// TwinCAT 3 PLC project Untitled1
// ProgramVersion: 3.1.4024.0
// libraries:
//   CmpBitmapPool, * (System)
//   Tc2_Standard, * (Beckhoff Automation GmbH)
//   Tc2_System, * (Beckhoff Automation GmbH)
//   Tc3_Module, * (Beckhoff Automation GmbH)
//   VisuDialogs, * (System)
// project tree:
//   / GlobalTextList.TcGTLO, PlcTask.TcTTO, Visualization Manager.TcVMO (not stored)
//   GVLs/ GVL_hesapSayfa.TcGVL, GVL_Mesai_Ucret.TcGVL, GVL_uye_panel.TcGVL, GVL_mesai_gun.TcGVL, GVL_mesai_saat.TcGVL, GVL_personel_kayit.TcGVL
//   POUs/ ImagePool.TcIPO (not stored), MAIN.TcPOU, POU_2.TcPOU
//   VISUs/ Hesap_Sayfa.TcVIS, Kayit_Sayfa.TcVIS, mesaigunleri_sayfa.TcVIS, MesaiSaat_sayfa.TcVIS, uyelik_sayfa.TcVIS, Ana_Sayfa.TcVIS
// real-time tasks:
//   TASK PlcTask: cycle T#10ms, priority 20, ADS port 350

CONFIGURATION Untitled1
    RESOURCE PLC ON TwinCAT3
        TASK PlcTask(INTERVAL := T#10ms, PRIORITY := 20);
        PROGRAM MAIN WITH PlcTask : MAIN;
    END_RESOURCE
END_CONFIGURATION

// ---- GVLs/GVL_hesapSayfa.TcGVL
{attribute 'qualified_only'}
VAR_GLOBAL
	

saydir1: TON;
start:BOOL;
cikis:BOOL;
gecensure:TIME;
gecenzaman:INT;
hesaplama:INT;






END_VAR

// ---- GVLs/GVL_Mesai_Ucret.TcGVL
{attribute 'qualified_only'}
VAR_GLOBAL
	

hesapla:INT;
mesaiUcret:INT;
online:BOOL;
kaydet:BOOL;






END_VAR

// ---- GVLs/GVL_uye_panel.TcGVL
{attribute 'qualified_only'}
VAR_GLOBAL
	








END_VAR

// ---- GVLs/GVL_mesai_gun.TcGVL
{attribute 'qualified_only'}
VAR_GLOBAL
	
pazartesi:BOOL;
sali:BOOL;
carsamba:BOOL;
persembe:BOOL;
cuma:BOOL;
cumartesi:BOOL;
pazar:BOOL;
kaydet:BOOL;


END_VAR

// ---- GVLs/GVL_mesai_saat.TcGVL
{attribute 'qualified_only'}
VAR_GLOBAL
	

kaydet:BOOL;
i:INT;
baslangicDk:INT;
bitisDk:INT;
baslangicSn:INT;
bitisSn:INT;
cikis:BOOL;
sayac:INT;
sayac1:INT;
j:INT;
sayac2:INT;
n:INT;
sayac3:INT;
h:INT;
mesaiucret:INT;
saat:INT;
mesaiSaaat:INT;



x1_mesaiSaat:INT;
x1_5mesaiSaat:REAL;
x_3mesaiSaat:REAL;
tum_mesai:REAL;




x1_5baslangicSaat : INT;
x_3baslangicSaat:INT;




x1bslangicSaat:INT;
x1bslangicdakika:INT;
x1bitisSaat:INT;
x1bitisdakika:INT;



x1_5bslangicSaat:INT;
x1_5bslangicdakika:INT;
x1_5bitisSaat:INT;
x1_5bitisdakika:INT;




x3bslangicSaat:INT;
x3bslangicdakika:INT;
x3bitisSaat:INT;
x3bitisdakika:INT;










baslangicdakika: STRING;
baslangicsaat: STRING;
bitisdakika: STRING;
bitissaat: STRING;




a:BOOL;
b:BOOL;
c:BOOL;
d:BOOL;
e:BOOL;
f:BOOL;






































END_VAR

// ---- GVLs/GVL_personel_kayit.TcGVL
{attribute 'qualified_only'}
VAR_GLOBAL
	

perid:STRING;
perisim:STRING;
perSoyisim:STRING;

perMesaiGun:BOOL;
perMesaiSaat:BOOL;

kaydet:BOOL;
msgtype:MESSAGEBOXDIALOG_TYPES;
messagetitle:STRING;
messagetext:STRING;
cikis3:BOOL;
sayac:INT;
i:INT := 1;
sayac1:INT;
j:INT;
sayac2:INT;
g:INT;



dogru : BOOL;
invisibleKayit : BOOL;





personelisim:ARRAY[1..70] OF STRING;
personelsoyisim:ARRAY[1..70] OF STRING;
personelid:ARRAY[1..70] OF STRING;






saydirici:R_TRIG ;



temizle:BOOL;
















END_VAR

// ---- POUs/MAIN.TcPOU
PROGRAM MAIN
VAR
	



isim:ARRAY[0..70] OF STRING;
kullanici: ARRAY[0..70] OF STRING;
sifreler: ARRAY[0..70] OF STRING;
soyisim:ARRAY[0..70] OF STRING;
gunler:ARRAY[1..7] OF BOOL;

ad:STRING;
soyad:STRING;
kuladi:STRING;
sifre:STRING;

kaydet:BOOL;







uyelik:BOOL;
uyelik1:BOOL;
sayici:INT;



giris:BOOL;




yenikul:STRING;
yenisifre:STRING;





msgtype:MESSAGEBOXDIALOG_TYPES;
msgtitle:STRING;
msgtxt:STRING;



i: INT;
j:INT;
	
	cikis: BOOL;
	

	

	saydir: R_TRIG;
	cikis2: BOOL;
	sayici1: INT;
	kaydet2: BOOL;
	sayici2: INT;
	g: INT;
	sayici3: INT;
	h: INT;
	n: INT;
	giris1: BOOL;
	
	mesai_saat_saydirici: R_TRIG;
	
END_VAR



msgtitle:='İşlem Durumu ';
msgtxt:='Kayıt İşlemi Başarılı..';


GVL_personel_kayit.messagetext:='Kayıt İşlemi Başarılı.. Mesai Ücreti Hesaplamak Mesai Günü Seç  Butonuna Basınız.';
GVL_personel_kayit.messagetitle:='Kayıt İşlemi Durumu';






Giris_Panel();
uyelik_panel();
Kayit_Sayfa();
mesai_gun();
mesai_saat();
Hesap_Panel();

ACTION Giris_Panel:

giris1:=FALSE;

IF GVL_personel_kayit.perMesaiGun THEN
	GVL_personel_kayit.dogru:=TRUE;
	
END_IF


IF giris=TRUE THEN
	
FOR n:=1 TO 70 BY 1 DO
	
  IF kullanici[n]=kuladi AND sifreler[n]=sifre AND NOT GVL_personel_kayit.dogru THEN
	  
 
	  VisuElems.CurrentVisu := 'Kayit_Sayfa';
	  
	  
	  
	 
  END_IF

  	
END_FOR

	
END_IF
END_ACTION

ACTION Hesap_Panel:

GVL_mesai_saat.mesaiucret:=50;
GVL_hesapSayfa.saydir1(IN:=GVL_hesapSayfa.start , PT:=T#10S , Q=>GVL_hesapSayfa.cikis , ET=>GVL_hesapSayfa.gecensure );

GVL_hesapSayfa.start:=TRUE;



IF GVL_hesapSayfa.cikis=TRUE THEN
	
 IF 
	 GVL_mesai_gun.pazartesi=TRUE  OR  GVL_mesai_gun.sali=TRUE OR  GVL_mesai_gun.carsamba=TRUE OR  GVL_mesai_gun.persembe=TRUE OR  GVL_mesai_gun.cuma=TRUE THEN
	
	
(*   IF GVL_mesai_saat.baslangicsaat < GVL_mesai_saat.bitissaat  THEN
    	GVL_hesapSayfa.hesaplama:= GVL_mesai_saat.bitissaat-GVL_mesai_saat.baslangicsaat;
		ELSE			
		GVL_hesapSayfa.hesaplama:=GVL_mesai_saat.baslangicsaat-GVL_mesai_saat.bitisdakika;
		
 
 
END_IF
 *)
	
	
	
 
 END_IF
 
 
 
 

 
(*  IF GVL_mesai_gun.cumartesi OR GVL_mesai_gun.pazar THEN
	 	
   	 
 GVL_hesapSayfa.hesaplama:= GVL_mesai_saat.bitisdakika-GVL_mesai_saat.baslangicdakika;
 
 
 END_IF
 *)
 
 
 



	
END_IF
END_ACTION

ACTION Kayit_sayfa:


GVL_personel_kayit.saydirici(CLK:=GVL_personel_kayit.kaydet , Q=>GVL_personel_kayit.cikis3 );

IF GVL_personel_kayit.kaydet THEN
	GVL_personel_kayit.invisibleKayit:=TRUE;
END_IF

IF VisuElems.CurrentVisu='mesaigunleri_sayfa'THEN
	GVL_personel_kayit.invisibleKayit:=FALSE;
END_IF


IF GVL_personel_kayit.kaydet=TRUE THEN
	
IF GVL_personel_kayit.cikis3=TRUE THEN
 
GVL_personel_kayit.sayac:=GVL_personel_kayit.sayac +1;

END_IF



FOR GVL_personel_kayit.i:=1 TO 70 BY 1 DO
	
IF GVL_personel_kayit.personelisim[GVL_personel_kayit.i] ='' THEN
	GVL_personel_kayit.personelisim[GVL_personel_kayit.i]:=GVL_personel_kayit.perisim;
		
ELSE
	GVL_personel_kayit.personelisim[GVL_personel_kayit.sayac]:=GVL_personel_kayit.perisim;
	
END_IF

EXIT;
END_FOR






IF GVL_personel_kayit.cikis3=TRUE THEN
	
	GVL_personel_kayit.sayac1:=GVL_personel_kayit.sayac1+1;		
END_IF

FOR GVL_personel_kayit.j:=1 TO 70 BY  1 DO
	
IF GVL_personel_kayit.personelsoyisim[GVL_personel_kayit.j]='' THEN
	GVL_personel_kayit.personelsoyisim[GVL_personel_kayit.j]:=GVL_personel_kayit.perSoyisim;
	ELSE
		GVL_personel_kayit.personelsoyisim[GVL_personel_kayit.sayac]:=GVL_personel_kayit.perSoyisim;
	
END_IF

EXIT;

END_FOR



IF GVL_personel_kayit.cikis3=TRUE THEN
	GVL_personel_kayit.sayac2:=GVL_personel_kayit.sayac2 +1;
	
END_IF

FOR GVL_personel_kayit.g:=1 TO 70 BY 1 DO
	
	IF GVL_personel_kayit.personelid[GVL_personel_kayit.g]='' THEN
		GVL_personel_kayit.personelid[GVL_personel_kayit.g]:=GVL_personel_kayit.perid;
		ELSE
		GVL_personel_kayit.personelid[GVL_personel_kayit.sayac2]:=GVL_personel_kayit.perid;	
		
	END_IF
	EXIT;
	
END_FOR



















END_IF




IF GVL_personel_kayit.temizle=TRUE THEN
	GVL_personel_kayit.perisim:='';
	GVL_personel_kayit.perSoyisim:='';
	GVL_personel_kayit.perid:='';
	
	
	
	


END_IF
END_ACTION

ACTION mesai_gun:





IF GVL_mesai_gun.pazartesi=TRUE THEN
	
	
GVL_mesai_gun.sali:=FALSE;
GVL_mesai_gun.carsamba:=FALSE;
GVL_mesai_gun.persembe:=FALSE;
GVL_mesai_gun.cuma:=FALSE;
GVL_mesai_gun.cumartesi:=FALSE;
GVL_mesai_gun.pazar:=FALSE;


END_IF






IF GVL_mesai_gun.sali=TRUE THEN
	
	
GVL_mesai_gun.pazartesi:=FALSE;
GVL_mesai_gun.carsamba:=FALSE;
GVL_mesai_gun.persembe:=FALSE;
GVL_mesai_gun.cuma:=FALSE;
GVL_mesai_gun.cumartesi:=FALSE;
GVL_mesai_gun.pazar:=FALSE;


END_IF





IF GVL_mesai_gun.carsamba=TRUE THEN
	
	
GVL_mesai_gun.pazartesi:=FALSE;
GVL_mesai_gun.sali:=FALSE;
GVL_mesai_gun.persembe:=FALSE;
GVL_mesai_gun.cuma:=FALSE;
GVL_mesai_gun.cumartesi:=FALSE;
GVL_mesai_gun.pazar:=FALSE;


END_IF




IF GVL_mesai_gun.persembe=TRUE THEN
	
	
GVL_mesai_gun.pazartesi:=FALSE;
GVL_mesai_gun.sali:=FALSE;
GVL_mesai_gun.carsamba:=FALSE;
GVL_mesai_gun.cuma:=FALSE;
GVL_mesai_gun.cumartesi:=FALSE;
GVL_mesai_gun.pazar:=FALSE;


END_IF





IF GVL_mesai_gun.cuma=TRUE THEN
	
	
GVL_mesai_gun.pazartesi:=FALSE;
GVL_mesai_gun.sali:=FALSE;
GVL_mesai_gun.carsamba:=FALSE;
GVL_mesai_gun.persembe:=FALSE;
GVL_mesai_gun.cumartesi:=FALSE;
GVL_mesai_gun.pazar:=FALSE;


END_IF






IF GVL_mesai_gun.cumartesi=TRUE THEN
	
	
GVL_mesai_gun.pazartesi:=FALSE;
GVL_mesai_gun.sali:=FALSE;
GVL_mesai_gun.carsamba:=FALSE;
GVL_mesai_gun.persembe:=FALSE;
GVL_mesai_gun.cuma:=FALSE;
GVL_mesai_gun.pazar:=FALSE;


END_IF
IF GVL_mesai_gun.pazar=TRUE THEN
	
	
GVL_mesai_gun.pazartesi:=FALSE;
GVL_mesai_gun.sali:=FALSE;
GVL_mesai_gun.carsamba:=FALSE;
GVL_mesai_gun.persembe:=FALSE;
GVL_mesai_gun.cumartesi:=FALSE;
GVL_mesai_gun.cuma:=FALSE;


END_IF
END_ACTION

ACTION mesai_saat:



GVL_mesai_saat.a:=FALSE;
GVL_mesai_saat.b:=FALSE;
GVL_mesai_saat.c:=FALSE;




 // Başlangıç Dakikası
IF GVL_mesai_saat.kaydet=TRUE THEN
	

	 
  
	IF GVL_mesai_saat.x1bslangicSaat>GVL_mesai_saat.x1bitisSaat THEN
	
	GVL_mesai_saat.x1_mesaiSaat:=GVL_mesai_saat.x1bslangicSaat-GVL_mesai_saat.x1bitisSaat;
	GVL_mesai_saat.a:=TRUE;
	ELSE
		
	GVL_mesai_saat.x1_mesaiSaat:=GVL_mesai_saat.x1bitisSaat-GVL_mesai_saat.x1bslangicSaat;
	GVL_mesai_saat.b:=TRUE;
	
	END_IF
 



	IF GVL_mesai_saat.x1_5bslangicSaat>GVL_mesai_saat.x1_5bitisSaat THEN
	
	GVL_mesai_saat.x1_5mesaiSaat:=(GVL_mesai_saat.x1_5bslangicSaat-GVL_mesai_saat.x1_5bitisSaat)*1.5;
	GVL_mesai_saat.c:=TRUE;
	
	ELSE
		
	
	GVL_mesai_saat.x1_5mesaiSaat := (GVL_mesai_saat.x1_5bitisSaat-GVL_mesai_saat.x1_5bslangicSaat)*1.5;
	GVL_mesai_saat.d:=TRUE;
	
	END_IF


	
     
	 




	IF GVL_mesai_saat.x3bslangicSaat>GVL_mesai_saat.x3bitisSaat THEN
	
	GVL_mesai_saat.x_3mesaiSaat:=(GVL_mesai_saat.x3bslangicSaat-GVL_mesai_saat.x3bitisSaat)*3;
	GVL_mesai_saat.e:=TRUE;
	ELSE
		
	GVL_mesai_saat.x_3mesaiSaat:=(GVL_mesai_saat.x3bitisSaat-GVL_mesai_saat.x3bslangicSaat)*3;
	GVL_mesai_saat.f:=TRUE;
	
	END_IF
	
	
	
	
	
	IF GVL_mesai_saat.a=TRUE  OR GVL_mesai_saat.b=TRUE  THEN
		GVL_mesai_saat.mesaiSaaat:=GVL_mesai_saat.x1_mesaiSaat;
		
	END_IF
	
	
	
	(* IF GVL_mesai_saat.c=TRUE  OR GVL_mesai_saat.d=TRUE  THEN
		
		GVL_mesai_saat.mesaiSaaat:=GVL_mesai_saat.x1_5mesaiSaat;
	END_IF
	
	IF GVL_mesai_saat.e=TRUE OR GVL_mesai_saat.f=TRUE THEN
		
		GVL_mesai_saat.mesaiSaaat:=GVL_mesai_saat.x_3mesaiSaat;
	END_IF *)
	
	GVL_mesai_saat.tum_mesai:=(GVL_mesai_saat.x1_mesaiSaat+GVL_mesai_saat.x1_5mesaiSaat+GVL_mesai_saat.x_3mesaiSaat);
 
	
	
	


END_IF
END_ACTION

ACTION Mesai_Ucret_Panel:



GVL_Mesai_Ucret.online:=TRUE;
END_ACTION

ACTION uyelik_panel:


saydir(CLK:=kaydet , Q=>cikis );
		
		

IF kaydet=TRUE THEN




IF cikis=TRUE THEN
	sayici:=sayici+1;
END_IF

	FOR i:=1 TO 70 BY 1 DO
	
		IF isim[i]='' THEN			
			isim[i]:=ad;
		ELSE
			isim[sayici]:=ad;
		END_IF
		
		EXIT;
		
	END_FOR



IF cikis=TRUE THEN
	sayici1:=sayici1+1;
END_IF



FOR j:=1 TO 70 BY 1 DO
	
  IF soyisim[j]='' THEN
	  soyisim[j]:=soyad;
   ELSE
	soyisim[sayici1]:=soyad;
  END_IF


EXIT;
END_FOR










IF cikis=TRUE THEN
	sayici2:=sayici2+1;
	END_IF



FOR g:=1 TO 70 BY 1 DO
	
  IF kullanici[g]='' THEN
	  kullanici[g]:=yenikul;
	  ELSE
		  kullanici[sayici2]:=yenikul;
  END_IF


EXIT;
END_FOR







IF cikis=TRUE THEN
	sayici3:=sayici3+1;
	END_IF



FOR h:=1 TO 70 BY 1 DO
	
  IF sifreler[h]='' THEN
	  sifreler[h]:=yenisifre;
	  ELSE
		  sifreler[sayici3]:=yenisifre;
  END_IF


EXIT;
END_FOR


























	

END_IF
END_ACTION

END_PROGRAM

// ---- POUs/POU_2.TcPOU
PROGRAM POU_2
VAR
END_VAR

END_PROGRAM

// ---- GlobalTextList.TcGTLO
TEXTLIST GlobalTextList
  899 = '  '
  16 = '                          İsim:'
  1263 = '                   İsim:'
  435 = '                  İsim:'
  382 = '                İsim:'
  1202 = '             Soyisim:'
  479 = '            Soyisim:'
  1142 = '           Soyisim:'
  551 = '          Soyisim:'
  85 = '        Personel ID:'
  1102 = '       Personel ID:'
  510 = '      Personel ID:'
  1073 = '      Soyisim:'
  905 = '   Soyisim:'
  742 = '  Mesai Saati :'
  778 = '  Mesai Saati Seç'
  682 = ' Yeni Kullanıcı Adı :'
  954 = '%d'
  897 = '%d Saat Mesai Yapılmıştır'
  1058 = '%d Saat Mesai Yapılmıştır.'
  772 = '%d:%d'
  997 = '%ds'
  74 = '%s'
  388 = '%s:%s'
  62 = "%t[Son Güncelleme :'ddd MMM dd.MM.yy'at' HH:mm:ss]"
  507 = '-----------'
  528 = '------------------------'
  966 = '---------------------------'
  628 = '----------------------------'
  333 = '------------------------------'
  654 = '-----------------------------------'
  850 = '07:45'
  549 = '07:45/ 18:45'
  996 = '07:45/ 18:45 (X1)'
  963 = '07:45/ 18:45 (X1,5)'
  709 = '07:45/ 18:45 (X2)'
  404 = '07:45/ 18:45 (X2,5)'
  422 = '07:45/ 18:45 (X3)'
  728 = '0:%s'
  1004 = '1,5/X Mesai'
  1156 = '1/X Mesai'
  990 = '18:45/ 18:45 (X1)'
  1298 = '18:45/ 18:45 (X1,5)'
  471 = '18:45/ 23:45 (X1,5)'
  794 = '18:45/ 23:45 (X2)'
  1060 = '18:45/ 23:45 (X2,5)'
  900 = '23:45/ 07:45 (X2)'
  744 = '23:45/ 07:45 (X2,5)'
  436 = '23:45/ 07:45 (X3)'
  666 = '23:45/ 18:45 (X3)'
  885 = '23:45/07:45 (X3)'
  271 = '23:45/8:45 (X3)'
  892 = '3/X Mesai'
  919 = ':'
  653 = '@afşa'
  410 = 'Adı :'
  425 = 'Adınız           :'
  953 = 'Adınız       :'
  790 = 'Adınız   :'
  977 = 'Adınız  :'
  942 = 'Adınız :'
  176 = 'Afşa Robotik'
  1317 = 'Alacağı Ücret :'
  34 = 'Ana Sayfaya Dön'
  580 = 'ascascas'
  827 = 'asfqwfsvsdv'
  509 = 'Başlangıç :'
  773 = 'Başlangıç Saati :'
  1122 = 'Bilgilendirme'
  220 = 'Bitiş  Saati :'
  1442 = 'Bitiş :'
  817 = 'Bugünün Tarihni Giriniz :'
  252 = 'Bugünün Tariini Giriniz :'
  270 = 'Buugünün Tariini Giriniz :'
  683 = 'CUMA'
  325 = 'CUMARTESİ'
  241 = 'd'
  793 = 'G,n Sayfası'
  627 = 'Geriye Dön'
  1107 = 'Geriye Dön '
  318 = 'GERİYE DÖN'
  558 = 'Giriş'
  83 = 'Giriş Yap'
  994 = 'GroupBox'
  1049 = 'Gün Sayfası'
  301 = 'Gün Seç'
  1115 = 'Gün Çizelgesi'
  970 = 'GÜN ÇİZELGESİ'
  881 = 'GÜN/SAAT ÇİZELGESİ'
  984 = 'HAFTA SONU'
  965 = 'Hafta Sonu'
  323 = 'Hafta İçi'
  822 = 'HAFTA İÇİ'
  950 = 'Hesapla'
  472 = 'HESAPLANAN ÜCRET'
  860 = 'Isim :'
  546 = 'Kaydet'
  504 = 'KAYDET'
  501 = 'Kayıt Bilgisi'
  582 = 'Kullanıcı Adı'
  334 = 'Kullanıcı Adı :'
  995 = 'Label'
  188 = 'Mesai Gün Çizelgesi'
  39 = 'Mesai Günü'
  374 = 'Mesai Günü :'
  681 = 'Mesai Günü Seç'
  868 = 'Mesai Saati'
  298 = 'Mesai Saati :'
  918 = 'Mesai Saati : '
  281 = 'Mesai Saati Seç'
  788 = 'Mesai Saatini Giriniz :'
  256 = 'Mesai Ücreti'
  962 = 'Mesai Ücreti Hesapla'
  322 = 'MESAİ SAATİ UYGULAMASI'
  257 = 'OLUŞTUR'
  5 = 'PAZAR'
  819 = 'PAZARTESİ'
  293 = 'Personel Bilgileri'
  521 = 'Personel Bilgisi'
  799 = 'PERSONEL BİLGİSİ'
  514 = 'Personel ID:'
  752 = 'PERSONEL MESAİ TAKİP UYGULAMASI'
  129 = 'PERSONEL MESAİ-TAKİP'
  545 = 'Personel Soyisim :'
  512 = 'Personel İd'
  93 = 'Personel İd :'
  219 = 'Personel İsim :'
  731 = 'PERŞEMBE'
  140 = 'S'
  311 = 'saassacaxzc'
  506 = 'SALI'
  59 = 'sdasqwfqwf'
  508 = 'Soyadı :'
  810 = 'Soyadınız :'
  66 = 'Soyisim'
  847 = 'Soyisim :'
  910 = 'Soyisim:'
  581 = 'sOYİSİM:'
  336 = 'Temizle'
  20 = 'ullanıcı Adı :'
  1206 = 'x(1,5)'
  1002 = 'x(3)'
  655 = 'x1'
  1441 = 'x3'
  833 = 'YENİ KAYIT OLUŞTURMA'
  118 = 'YENİ ÜYE OLUŞTURMA'
  239 = 'Zamanı Giriniz :'
  476 = 'zxcZxc'
  299 = 'ÇARŞAMBA'
  452 = 'ÇIKIŞ'
  969 = 'Ücret :'
  602 = 'Üyelik Oluştur'
  937 = 'İsim      :'
  569 = 'İsim    :'
  614 = 'İsim  :'
  393 = 'İsim :'
  242 = 'İsim:'
  431 = 'Şifre'
  908 = 'Şifre :'
END_TEXTLIST

// ---- VISUs/Hesap_Sayfa.TcVIS
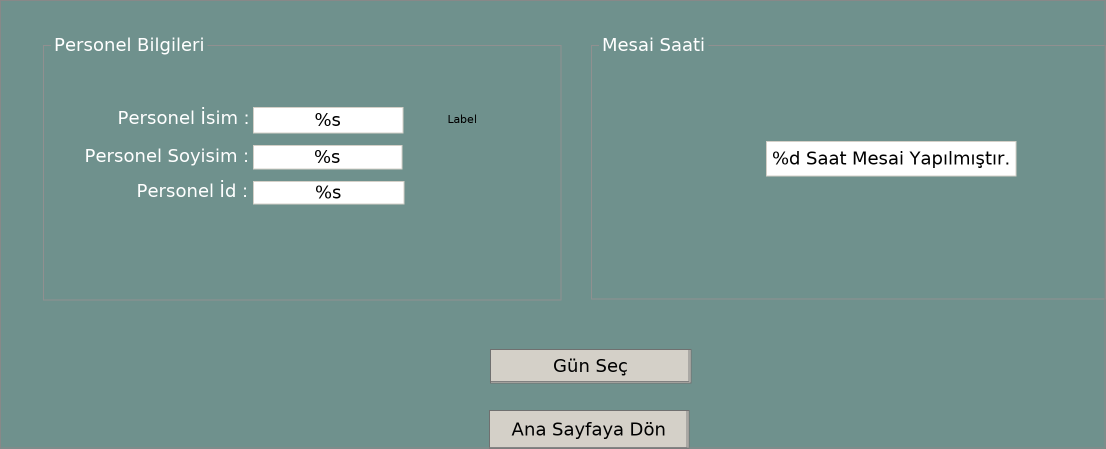
VISUALIZATION Hesap_Sayfa  // 1106x449
    GroupBox (43,37 518x263), "Personel Bilgileri"
        Label (69,66 143x30), "Personel İsim :"
        Label (44,104 160x30), "Personel Soyisim :"
        Label (78,139 143x30), "Personel İd :"
        Textfield (210,70 150x26), "%s", text variable: GVL_personel_kayit.perisim
        Textfield (210,108 149x24), "%s", text variable: GVL_personel_kayit.perSoyisim
        Textfield (210,144 151x23), "%s", text variable: GVL_personel_kayit.perid
    GroupBox (591,37 515x262), "Mesai Saati"
        Textfield (175,104 250x35), "%d Saat Mesai Yapılmıştır.", text variable: GVL_mesai_saat.tum_mesai
    Label (462,119 1x1), "Label"
    Button (490,349 201x34), "Gün Seç"
        OnMouseClick: change screen: mesaigunleri_sayfa
    Button (489,410 200x39), "Ana Sayfaya Dön"
        OnMouseClick: change screen: Ana_Sayfa
END_VISUALIZATION

// ---- VISUs/Kayit_Sayfa.TcVIS
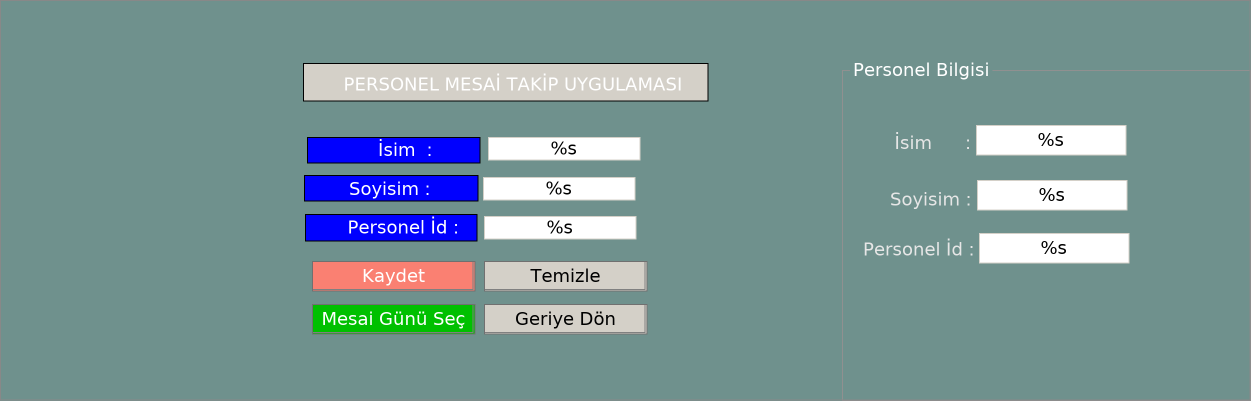
VISUALIZATION Kayit_Sayfa  // 1251x401
    Rectangle (305,214 172x27)
    Rectangle (303,63 405x38)
    Rectangle (307,137 173x26)
    Rectangle (304,175 174x26)
    Textfield (488,137 152x23), "%s", text variable: GVL_personel_kayit.perisim
        OnMouseClick: write the text variable via Edit
    Label (294,176 192x26), "Soyisim :"
    Label (323,132 165x36), "İsim :"
    Textfield (483,177 152x23), "%s", text variable: GVL_personel_kayit.perSoyisim
        OnMouseClick: write the text variable via Edit
    Label (315,71 396x27), "PERSONEL MESAİ TAKİP UYGULAMASI"
    Label (338,213 131x29), "Personel İd :"
    Textfield (484,216 152x23), "%s", text variable: GVL_personel_kayit.perid
        OnMouseClick: write the text variable via Edit
    Button (312,261 163x30), "Kaydet"
        tap GVL_personel_kayit.kaydet
        OnMouseClick: OpenDialog Dialog=VisuDialogs.MessageBox, Parameters={eType: GVL_personel_kayit.msgtype, sMessageTxt: GVL_personel_kayit.messagetext, sTitle: GVL_personel_kayit.messagetitle}, OpenModal=True, OpenCentered=True
    GroupBox (842,62 409x339), "Personel Bilgisi"
        Label (16,66 150x30), "İsim :"
        Label (14,123 150x29), "Soyisim :"
        Label (2,172 150x31), "Personel İd :"
        Textfield (135,118 150x30), "%s", text variable: GVL_personel_kayit.perSoyisim
            OnMouseClick: write the text variable via Edit
        Textfield (137,171 150x30), "%s", text variable: GVL_personel_kayit.perid
            OnMouseClick: write the text variable via Edit
        Textfield (134,63 150x30), "%s", text variable: GVL_personel_kayit.perisim
            OnMouseClick: write the text variable via Edit
    Button (312,304 163x30), "Mesai Günü Seç", invisible if: NOT GVL_personel_kayit.invisibleKayit
        tap GVL_personel_kayit.perMesaiGun
        OnMouseClick: change screen: mesaigunleri_sayfa
    Button (484,261 163x30), "Temizle"
        tap GVL_personel_kayit.temizle
    Button (484,304 163x30), "Geriye Dön"
        OnMouseClick: change screen: Ana_Sayfa
END_VISUALIZATION

// ---- VISUs/mesaigunleri_sayfa.TcVIS
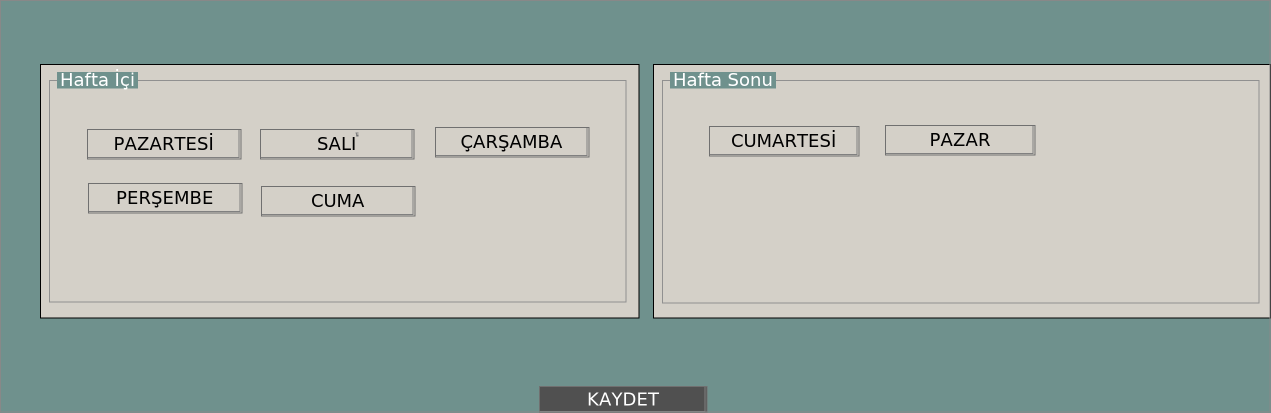
VISUALIZATION mesaigunleri_sayfa  // 1271x413
    Rectangle (653,64 618x254)
    Rectangle (40,64 599x254)
    GroupBox (49,72 577x230), "Hafta İçi"
        Button (38,57 154x30), "PAZARTESİ"
            toggle GVL_mesai_gun.pazartesi
        Button (211,57 154x30), "SALI"
            toggle GVL_mesai_gun.sali
        Button (386,55 154x30), "ÇARŞAMBA"
            toggle GVL_mesai_gun.carsamba
        Button (39,111 154x30), "PERŞEMBE"
            toggle GVL_mesai_gun.persembe
        Button (212,114 154x30), "CUMA"
            toggle GVL_mesai_gun.cuma
    GroupBox (662,72 597x231), "Hafta Sonu"
        Button (47,54 150x30), "CUMARTESİ"
            toggle GVL_mesai_gun.cumartesi
        Button (223,53 150x30), "PAZAR"
            toggle GVL_mesai_gun.pazar
    Button (539,386 168x27), "KAYDET"
        tap GVL_mesai_gun.kaydet
        OnMouseClick: change screen: MesaiSaat_sayfa
    Button (357,135 1x0)
END_VISUALIZATION

// ---- VISUs/MesaiSaat_sayfa.TcVIS
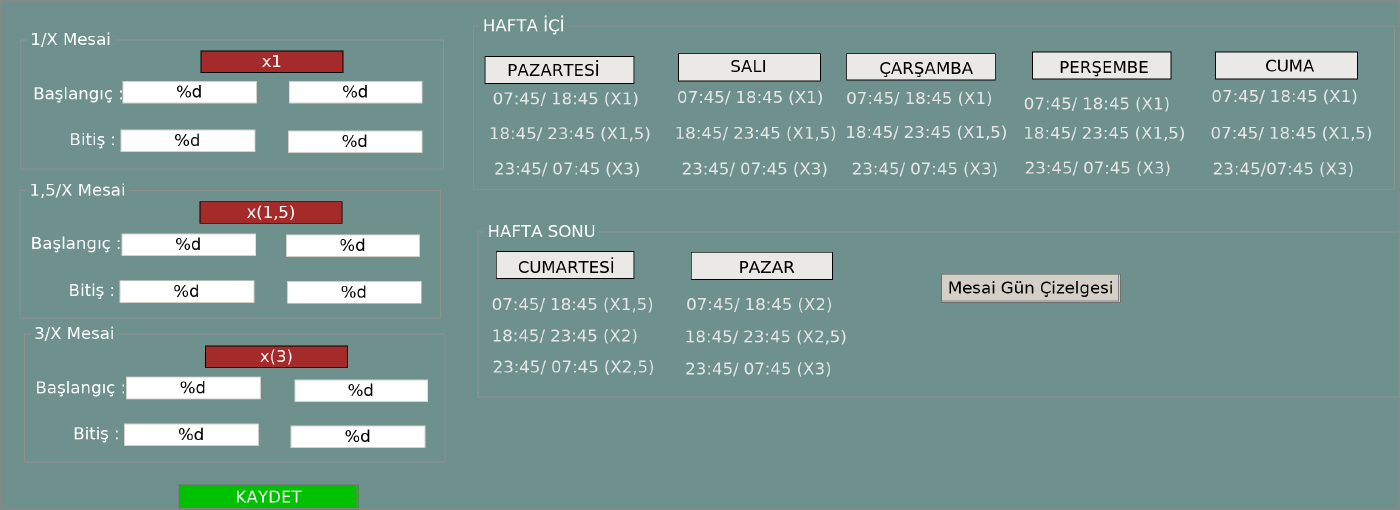
VISUALIZATION MesaiSaat_sayfa  // 1522x555
    Button (194,527 196x28), "KAYDET"
        toggle GVL_mesai_saat.kaydet
        OnMouseClick: change screen: Hesap_Sayfa
    Button (1023,298 195x31), "Mesai Gün Çizelgesi"
        OnMouseClick: change screen: gun_cizelge
    GroupBox (514,20 1002x186), "HAFTA İÇİ"
        Rectangle (807,36 155x30)
        Rectangle (608,36 151x30)
        Rectangle (406,38 162x29)
        Rectangle (223,38 155x30)
        Rectangle (13,41 162x30)
        Label (10,36 156x41), "PAZARTESİ"
        Label (227,28 146x49), "SALI"
        Label (414,32 159x45), "ÇARŞAMBA"
        Label (616,36 141x35), "PERŞEMBE"
        Label (818,30 141x44), "CUMA"
        Label (21,63 160x49), "07:45/ 18:45 (X1)"
        Label (21,101 169x49), "18:45/ 23:45 (X1,5)"
        Label (15,81 169x30)
        Label (217,71 169x30), "07:45/ 18:45 (X1)"
        Label (223,102 169x46), "18:45/ 23:45 (X1,5)"
        Label (401,72 169x30), "07:45/ 18:45 (X1)"
        Label (406,109 174x30), "18:45/ 23:45 (X1,5)"
        Label (594,78 169x30), "07:45/ 18:45 (X1)"
        Label (595,110 183x30), "18:45/ 23:45 (X1,5)"
        Label (798,70 169x30), "07:45/ 18:45 (X1)"
        Label (802,110 176x30), "07:45/ 18:45 (X1,5)"
        Label (797,149 169x30), "23:45/07:45 (X3)"
        Label (595,148 169x30), "23:45/ 07:45 (X3)"
        Label (407,149 169x30), "23:45/ 07:45 (X3)"
        Label (222,149 169x30), "23:45/ 07:45 (X3)"
        Label (18,149 169x30), "23:45/ 07:45 (X3)"
    GroupBox (519,244 1003x188), "HAFTA SONU"
        Rectangle (20,29 150x30)
        Label (20,32 154x30), "CUMARTESİ"
        Rectangle (232,30 154x30)
        Label (231,28 167x38), "PAZAR"
        Label (16,63 175x49), "07:45/ 18:45 (X1,5)"
        Label (15,98 160x47), "18:45/ 23:45 (X2)"
        Label (219,63 175x49), "07:45/ 18:45 (X2)"
        Label (228,98 171x49), "18:45/ 23:45 (X2,5)"
        Label (212,133 187x49), "23:45/ 07:45 (X3)"
    Label (535,375 177x49), "23:45/ 07:45 (X2,5)"
    GroupBox (22,35 460x149), "1/X Mesai"
        Textfield (111,53 146x24), "%d", text variable: GVL_mesai_saat.x1bslangicSaat
            OnMouseClick: write the text variable via VisuDialogs.Numpad, min 8, max 19
        Textfield (292,53 145x24), "%d", text variable: GVL_mesai_saat.x1bslangicdakika
            OnMouseClick: write the text variable via VisuDialogs.Numpad, min 0, max 59
        Textfield (109,106 146x24), "%d", text variable: GVL_mesai_saat.x1bitisSaat
            OnMouseClick: write the text variable via VisuDialogs.Numpad, min 8, max 19
        Textfield (291,107 146x24), "%d", text variable: GVL_mesai_saat.x1bitisdakika
            OnMouseClick: write the text variable via VisuDialogs.Numpad, min 0, max 59
        Rectangle (196,20 155x24), "x1"
        Label (4,102 150x30), "Bitiş :"
    Label (14,87 143x30), "Başlangıç :"
    GroupBox (21,199 458x147), "1,5/X Mesai"
        Textfield (111,55 146x24), "%d", text variable: GVL_mesai_saat.x1_5bslangicSaat
            OnMouseClick: write the text variable via VisuDialogs.Numpad, min 19, max 23
        Textfield (290,56 145x24), "%d", text variable: GVL_mesai_saat.x1_5bslangicdakika
            OnMouseClick: write the text variable via VisuDialogs.Numpad, min 0, max 59
        Textfield (109,106 146x24), "%d", text variable: GVL_mesai_saat.x1_5bitisSaat
            OnMouseClick: write the text variable via VisuDialogs.Numpad, min 19, max 23
        Textfield (291,107 146x24), "%d", text variable: GVL_mesai_saat.x1_5bitisdakika
            OnMouseClick: write the text variable via VisuDialogs.Numpad, min 0, max 59
        Label (4,102 150x30), "Bitiş :"
        Rectangle (196,20 155x24), "x(1,5)"
    Label (8,250 150x30), "Başlangıç :"
    GroupBox (26,355 458x148), "3/X Mesai"
        Textfield (111,55 146x24), "%d", text variable: GVL_mesai_saat.x3bslangicSaat
            OnMouseClick: write the text variable via VisuDialogs.Numpad
        Textfield (294,58 145x24), "%d", text variable: GVL_mesai_saat.x3bslangicdakika
            OnMouseClick: write the text variable via VisuDialogs.Numpad, min 45
        Textfield (109,106 146x24), "%d", text variable: GVL_mesai_saat.x3bitisSaat
            OnMouseClick: write the text variable via VisuDialogs.Numpad
        Textfield (290,108 146x24), "%d", text variable: GVL_mesai_saat.x3bitisdakika
            OnMouseClick: write the text variable via VisuDialogs.Numpad
        Label (4,102 150x30), "Bitiş :"
        Rectangle (197,21 155x24), "x(3)"
    Label (13,407 150x30), "Başlangıç :"
END_VISUALIZATION

// ---- VISUs/uyelik_sayfa.TcVIS
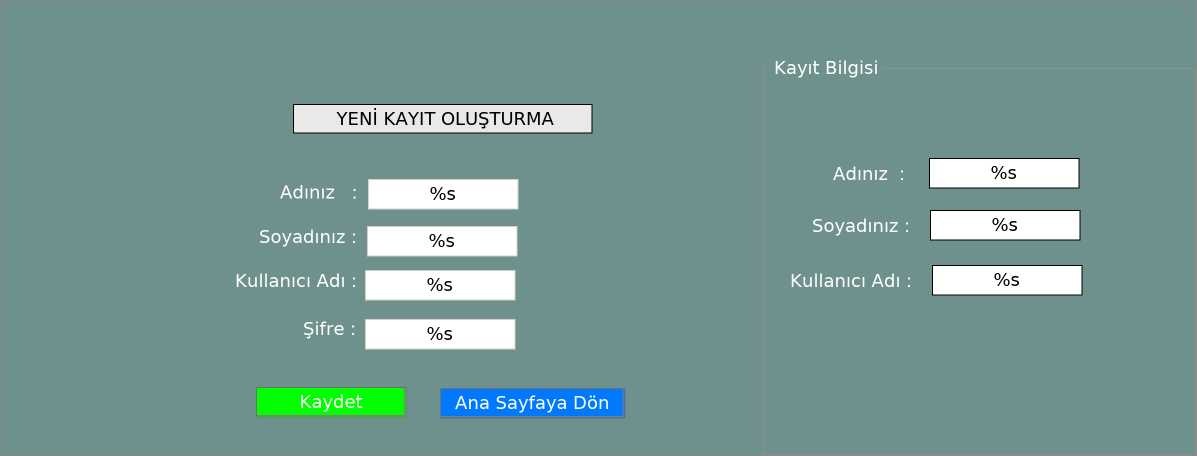
VISUALIZATION uyelik_sayfa  // 1197x456
    Rectangle (293,104 299x29)
    Label (244,176 150x33), "Adınız :"
    Label (233,222 150x30), "Soyadınız :"
    Label (216,265 160x32), "Kullanıcı Adı :"
    Label (255,315 149x28), "Şifre :"
    Label (311,104 269x30), "YENİ KAYIT OLUŞTURMA"
    Textfield (368,179 150x30), "%s", text variable: MAIN.ad
        OnMouseClick: write the text variable via Edit
    Textfield (367,226 150x30), "%s", text variable: MAIN.soyad
        OnMouseClick: write the text variable via Edit
    Textfield (365,319 150x30), "%s", text variable: MAIN.yenisifre
        OnMouseClick: write the text variable via Edit
    Textfield (365,270 150x30), "%s", text variable: MAIN.yenikul
        OnMouseClick: write the text variable via Edit
    Button (256,387 150x30), "Kaydet"
        tap MAIN.kaydet
        OnMouseClick: OpenDialog Dialog=VisuDialogs.MessageBox, Parameters={eType: MAIN.msgtype, sMessageTxt: MAIN.msgtxt, sTitle: MAIN.msgtitle}, OpenModal=True, OpenCentered=True
    Button (440,388 185x30), "Ana Sayfaya Dön"
        OnMouseClick: change screen: Ana_Sayfa
    GroupBox (763,60 434x396), "Kayıt Bilgisi"
        Rectangle (166,98 150x30), "%s", text variable: MAIN.ad
        Label (38,99 136x30), "Adınız :"
        Label (23,151 150x30), "Soyadınız :"
        Rectangle (167,150 150x30), "%s", text variable: MAIN.soyad
        Label (13,206 150x30), "Kullanıcı Adı :"
        Rectangle (169,205 150x30), "%s", text variable: MAIN.yenikul
END_VISUALIZATION

// ---- VISUs/Ana_Sayfa.TcVIS
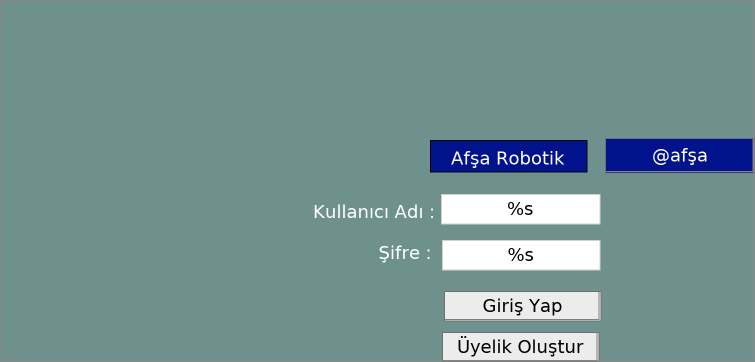
VISUALIZATION Ana_Sayfa  // 755x362
    Rectangle (430,140 157x32)
    Label (299,197 150x30), "Kullanıcı Adı :"
    Label (330,238 150x30), "Şifre :"
    Textfield (441,194 159x30), "%s", text variable: MAIN.kuladi
        OnMouseClick: write the text variable via Edit
    Textfield (442,240 158x30), "%s", text variable: MAIN.sifre
        OnMouseClick: write the text variable via Edit, password
    Button (444,291 157x30), "Giriş Yap"
        tap MAIN.giris
    Button (442,332 157x30), "Üyelik Oluştur"
        tap MAIN.uyelik
        OnMouseClick: change screen: uyelik_sayfa
    Label (288,144 440x29), "Afşa Robotik"
    Button (605,138 150x35), "@afşa", invisible if: MAIN.giris1
        tap MAIN.giris1
        OnMouseClick: change screen: uyelik_sayfa
END_VISUALIZATION
